TYPE ST_NeedleRemoveAllocate :
STRUCT
	Info 	: ST_NeedleAllocateinfo;
END_STRUCT
END_TYPE

(* stored: Version 1.1.0.1, ProductVersion 3.1.4024.13
   DUT ST_NeedleRemoveAllocate: Id {4bfc01a1-ebf9-421c-b8fc-3258f5dd2dc9} *)
